(* LS Electric XG5000 project: DataConversion_Example *)
(* PLC LSPLC *)
(* module base 0 slot 0: Input/Output Module:XEM-DN/DP32HP (DC 24V Input, Transistor Output, 32 Contacts) *)
(* module base 0 slot 1: Internal Positioning:XBF-PO06E (Open Collector Type, 6 Axis) *)
(* module base 0 slot 2: EtherNet/IP:XBL-EIPT (EtherNet/IP communication module, electrical) *)

(* Comments on direct variables
%IX0.0.0	this is comment 1
*)

PROGRAM DirectMemory_Example (* task: Scan Program *)
VAR
    GS20_BYTE_Input AT %MB0 : ARRAY[0..31] OF BYTE; (* T2O input data for GS20 in bytes *)
    GS20_BYTE_Output AT %MB32 : ARRAY[0..5] OF BYTE; (* O2T output data for GS20 in bytes *)
    GS20_DWORD_Input AT %MD0 : ARRAY[0..7] OF DWORD; (* Conversion of input data to DWORD data type *)
    GS20_WORD_Input AT %MW0 : ARRAY[0..15] OF WORD; (* Conversion of input data to WORD data type *)
    GS20_WORD_Output AT %MW16 : ARRAY[0..2] OF WORD; (* Conversion of output data to WORD data type. *)
END_VAR

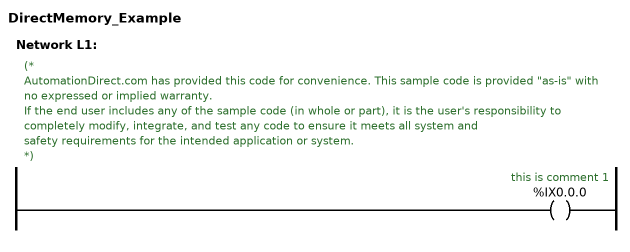
(* ( * / AutomationDirect.com has provided this code for convenience. This sample code is provided "as-is" with no expressed or implied warranty. / If the end user includes any of the sample code (in whole or part), it is the user's responsibility to completely modify, integrate, and test any code to ensure it meets all system and / safety requirements for the intended application or system. / * ) *)
(* Rung L1 *)
%IX0.0.0 := TRUE;
END_PROGRAM

PROGRAM DataConversion_Functions_LD (* task: Scan Program *)
VAR
    DwordLocation : INT; (* for loop variable *)
    GS20_BYTE_Input : ARRAY[0..31] OF BYTE; (* T2O input data for GS20 in bytes *)
    GS20_BYTE_Output : ARRAY[0..5] OF BYTE; (* O2T output data for GS20 in bytes *)
    GS20_DWORD_Input : ARRAY[0..7] OF DWORD; (* Conversion of input data to DWORD data type *)
    GS20_WORD_Input : ARRAY[0..15] OF WORD; (* Conversion of input data to WORD data type *)
    GS20_WORD_Output : ARRAY[0..2] OF WORD; (* Conversion of output data to WORD data type. *)
    HighByte : INT; (* for loop variable *)
    LowByte : INT; (* for loop variable *)
    WordLocation : INT; (* for loop variable *)
END_VAR

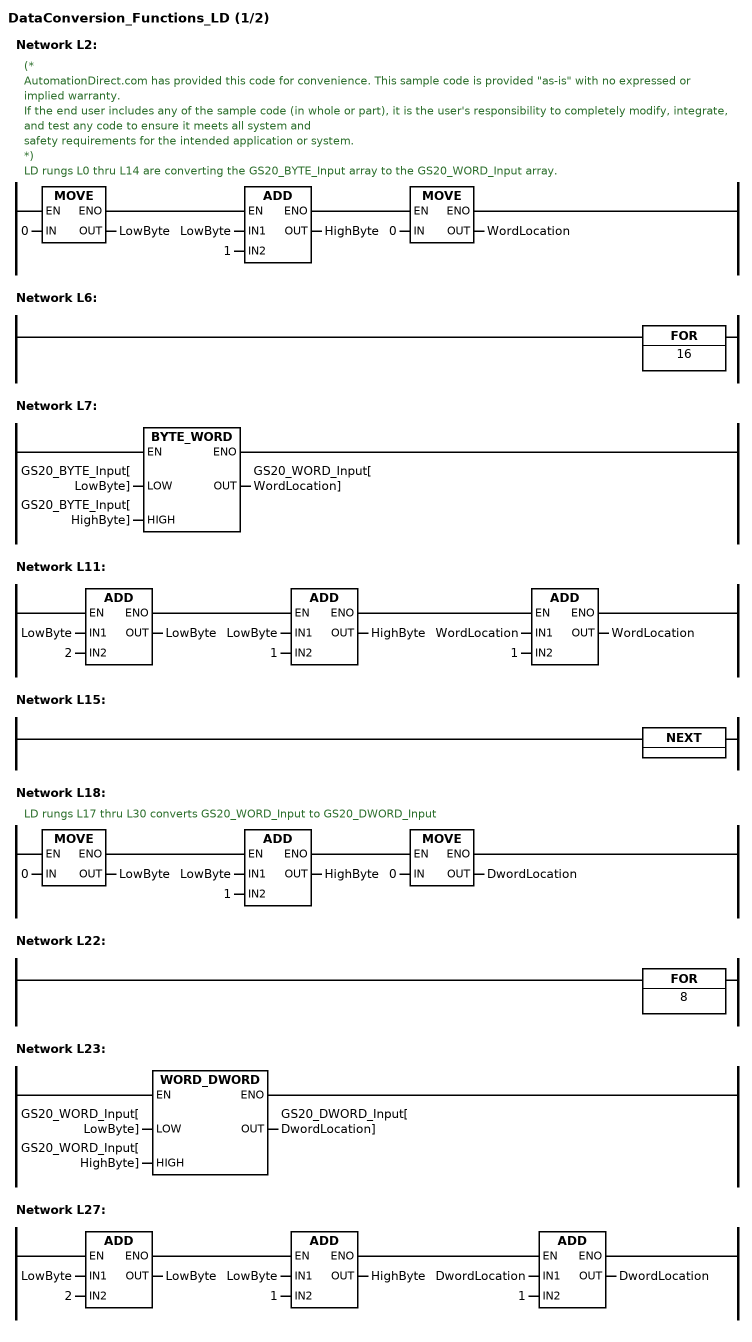
(* ( * / AutomationDirect.com has provided this code for convenience. This sample code is provided "as-is" with no expressed or implied warranty. / If the end user includes any of the sample code (in whole or part), it is the user's responsibility to completely modify, integrate, and test any code to ensure it meets all system and / safety requirements for the intended application or system. / * ) *)
(* LD rungs L0 thru L14 are converting the GS20_BYTE_Input array to the GS20_WORD_Input array. *)
(* Rung L2 *)
LowByte := 0;
HighByte := LowByte + 1;
WordLocation := 0;
(* Rung L6 *)
FOR(16);
(* Rung L7 *)
GS20_WORD_Input[WordLocation] := BYTE_WORD(LOW := GS20_BYTE_Input[LowByte], HIGH := GS20_BYTE_Input[HighByte]);
(* Rung L11 *)
LowByte := LowByte + 2;
HighByte := LowByte + 1;
WordLocation := WordLocation + 1;
(* Rung L15 *)
NEXT();
(* LD rungs L17 thru L30 converts GS20_WORD_Input to GS20_DWORD_Input *)
(* Rung L18 *)
LowByte := 0;
HighByte := LowByte + 1;
DwordLocation := 0;
(* Rung L22 *)
FOR(8);
(* Rung L23 *)
GS20_DWORD_Input[DwordLocation] := WORD_DWORD(LOW := GS20_WORD_Input[LowByte], HIGH := GS20_WORD_Input[HighByte]);
(* Rung L27 *)
LowByte := LowByte + 2;
HighByte := LowByte + 1;
DwordLocation := DwordLocation + 1;

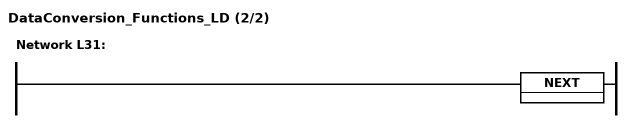
(* Rung L31 *)
NEXT();
END_PROGRAM

PROGRAM DataConversion_Functions_ST (* task: Scan Program *)
VAR
    DwordLocation : INT; (* for loop variable *)
    GS20_BYTE_Input : ARRAY[0..31] OF BYTE; (* T2O input data for GS20 in bytes *)
    GS20_BYTE_Output : ARRAY[0..5] OF BYTE; (* O2T output data for GS20 in bytes *)
    GS20_DWORD_Input : ARRAY[0..7] OF DWORD; (* Conversion of input data to DWORD data type *)
    GS20_WORD_Input : ARRAY[0..15] OF WORD; (* Conversion of input data to WORD data type *)
    GS20_WORD_Output : ARRAY[0..2] OF WORD; (* Conversion of output data to WORD data type. *)
    HighByte : INT; (* for loop variable *)
    i : INT; (* for loop variable *)
    LowByte : INT; (* for loop variable *)
    WordLocation : INT; (* for loop variable *)
END_VAR
(* 
AutomationDirect.com has provided this code for convenience. This sample code is provided "as-is" with no expressed or implied warranty. 
 If the end user includes any of the sample code (in whole or part), it is the user's responsibility to completely modify, integrate, and test any code to ensure it meets all system and 
 safety requirements for the intended application or system.
 *)
(* Convert GS20_BYTE_Input to GS20_WORD_Input *)
LowByte := 0;
HighByte := LowByte +1;
WordLocation := 0;

FOR i:=0 TO 15 BY 1 DO
	
	GS20_WORD_Input[WordLocation] := BYTE_WORD(LOW:=GS20_BYTE_Input[LowByte], HIGH:=GS20_BYTE_Input[HighByte]);
	
	LowByte := LowByte + 2;
	HighByte := LowByte +1;
	WordLocation := WordLocation + 1;
END_FOR;

(* Convert GS20_WORD_Input to GS20_DWORD_Input *)
LowByte := 0;
HighByte := LowByte +1;
DwordLocation := 0;

FOR i:=0 TO 7 BY 1 DO
	
	GS20_DWORD_Input[DwordLocation] := WORD_DWORD(LOW:=GS20_WORD_Input[LowByte], HIGH:=GS20_WORD_Input[HighByte]);
	
	LowByte := LowByte + 2;
	HighByte := LowByte +1;
	DwordLocation := DwordLocation + 1;
END_FOR;
END_PROGRAM